LIN {X 0,Y 22.752,Z 513.068,A -85,B 0,C 180,E1 -32130,E2 -32130} C_VEL
LIN {X 0,Y 21.649,Z 513.101,A -85,B 0,C 180,E1 -32116.864,E2 -32116.864} C_VEL
LIN {X 0,Y 21.546,Z 515.1,A -85,B 0,C 180,E1 -32111.597,E2 -32111.597} C_VEL
LIN {X 0,Y 21.546,Z 600,A -85,B 0,C 180,E1 -32111.597,E2 -32111.597} C_VEL
LIN {X 0,Y 21.546,Z 600,A -85,B 0,C 180,E1 -32111.597,E2 -32111.597}

QRS_NEXT_CUT()

QRS_NEXT()
QRS_HOME()

END
